PROGRAM MAIN
VAR
END_VAR

END_PROGRAM

(* stored: Version 1.1.0.1
   POU MAIN: Id {46c6155e-1631-4f07-9de1-af6d71d4f845} *)
